// TIA Portal V18 export
DATA_BLOCK "AHURegulators"   // DB105
{ S7_Optimized_Access := 'FALSE' }
VERSION : 0.1
// stored: AutoNumber false, DBAccessibleFromOPCUA true, IsOnlyStoredInLoadMemory false, IsWriteProtectedInAS false
   VAR RETAIN
      Regulators { S7_SetPoint := 'True'} : "UDT_AHUsRegulators";
   END_VAR
BEGIN
   Regulators.Cfg.cTempHeating[1] := 2;
   Regulators.FreshAirCoef.IAQ[1..3] := 0.2;
   Regulators.FreshAirCoef.BuildingdP[1..3] := 0.2;
END_DATA_BLOCK
